(* IEC 61131-3 sources: teller/JD_Teller_LC2_V11/Class/JD_OR_Teller, 1 file *)

(* ---- JD_OR_Teller.st ---- *)
(*!
<Class
	Name               = "JD_OR_Teller"
	Revision           = "1.0"
	RealtimeTask       = "false"
	CyclicTask         = "false"
	BackgroundTask     = "false"
	Sigmatek           = "false"
	OSInterface        = "false"
	HighPriority       = "false"
	Automatic          = "false"
	UpdateMode         = "Prescan"
	SharedCommandTable = "true"
	Objectsize         = "(284,120)">
	<Channels>
		<Server Name="ClassSvr" Visualized="false" Initialize="false" WriteProtected="true" Retentive="false"/>
		<Server Name="In1" Visualized="false" Initialize="false" WriteProtected="false" Retentive="false"/>
		<Server Name="In2" Visualized="false" Initialize="false" WriteProtected="false" Retentive="false"/>
		<Client Name="Out" Required="true" Internal="false"/>
	</Channels>
	<RevDoku>
		<Owner Company="JD" Author="SV"/>
		<Dokumentation Revision="1.1" Date="2014-09-04" Author="SV" Company="JD" Description="Kopie van JD_OR rev 1.2.  Init toegevoegd die een nul schrijft op server In1"/>
	</RevDoku>
</Class>
*)
JD_OR_Teller : CLASS
  //Servers:
	ClassSvr 	: SvrChCmd_DINT;
	In1 	: SvrCh_DINT;
	In2 	: SvrCh_DINT;
  //Clients:
	Out 	: CltCh_DINT;
  //Variables:
  //Functions:

	FUNCTION VIRTUAL GLOBAL Init;

	FUNCTION VIRTUAL GLOBAL In1::Write
		VAR_INPUT
			input (EAX) 	: DINT;
		END_VAR
		VAR_OUTPUT
			result (EAX) 	: DINT;
		END_VAR;

	FUNCTION VIRTUAL GLOBAL In2::Write
		VAR_INPUT
			input (EAX) 	: DINT;
		END_VAR
		VAR_OUTPUT
			result (EAX) 	: DINT;
		END_VAR;
  //Tables:
	FUNCTION @STD
		VAR_OUTPUT
			ret_code	: CONFSTATES;
		END_VAR;
	FUNCTION GLOBAL TAB @CT_;
END_CLASS;

FUNCTION VIRTUAL GLOBAL JD_OR_Teller::Init

  if _FirstScan then
    In1.Write(input:=0);
  end_if;

END_FUNCTION

FUNCTION VIRTUAL GLOBAL JD_OR_Teller::In1::Write
	VAR_INPUT
		input (EAX) 	: DINT;
	END_VAR
	VAR_OUTPUT
		result (EAX) 	: DINT;
	END_VAR

	In1 := input;

  if  In1 = 1 | In2 = 1 then
      Out := 0;
      Out.Write(Out);
  else
      Out := 1;
      Out.Write(Out);
  end_if;

 	result := In1;

END_FUNCTION

FUNCTION VIRTUAL GLOBAL JD_OR_Teller::In2::Write
	VAR_INPUT
		input (EAX) 	: DINT;
	END_VAR
	VAR_OUTPUT
		result (EAX) 	: DINT;
	END_VAR

	In2 := input;

  if  In1 = 1 | In2 = 1 then
      Out := 0;
      Out.Write(Out);
  else
      Out := 1;
      Out.Write(Out);
  end_if;

 	result := In2;

END_FUNCTION
